TYPE ST_RegMapStorage :
STRUCT
    nStateOfCharge: WORD;
    nStorageAvailable: WORD;
    nVoltageInternal: WORD;
    nState: E_StorageChargeState;
    nSfStateOfCharge: WORD := INT_TO_UINT(-2);
END_STRUCT
END_TYPE

(* stored: Version 1.1.0.1
   DUT ST_RegMapStorage: Id {71e32fe8-7d97-476d-b94c-40cf3c24ad65} *)
